FUNCTION_BLOCK EQUIP_TRIManager (* Composite Function Block Type *)
  (* Standard: 61499-2 *)
  (* Version 0.0, 08/01/2026, Schneider Electric, template *)
  PACKAGE Main;
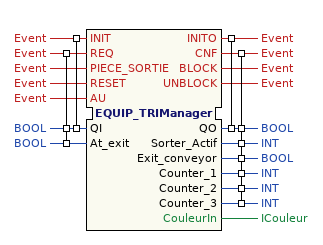
  EVENT_INPUT
    INIT WITH QI; (* Initialization Request *)
    REQ WITH QI, At_exit; (* Normal Execution Request *)
    PIECE_SORTIE;
    RESET; (* Reset compteurs et etapes *)
    AU; (* Arret urgence *)
  END_EVENT
  EVENT_OUTPUT
    INITO WITH QO; (* Initialization Confirm *)
    CNF WITH QO, Sorter_Actif, Exit_conveyor, Counter_1, Counter_2, Counter_3; (* Execution Confirmation *)
    BLOCK; (* Bloquer le convoyeur d'entrée *)
    UNBLOCK; (* Débloquer le convoyeur d'entrée *)
  END_EVENT
  VAR_INPUT
    QI : BOOL; (* Input event qualifier *)
    At_exit : BOOL; (* Capteur sortie - TRUE si piece presente *)
  END_VAR
  VAR_OUTPUT
    QO : BOOL; (* Output event qualifier *)
    Sorter_Actif : INT;
    Exit_conveyor : BOOL;
    Counter_1 : INT;
    Counter_2 : INT;
    Counter_3 : INT;
  END_VAR
  PLUGS
    CouleurIn : ICouleur; (* Entrée couleur *)
  END_PLUGS
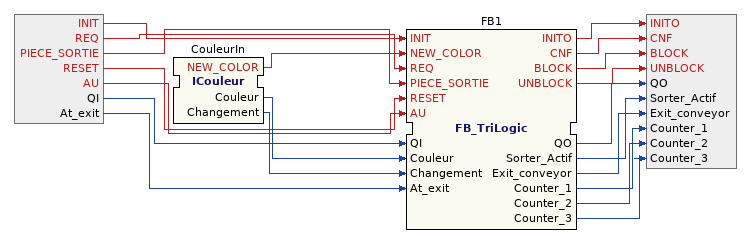
  FBS
    FB1 : FB_TriLogic;
  END_FBS
  EVENT_CONNECTIONS
    FB1.INITO TO INITO;
    FB1.CNF TO CNF;
    FB1.BLOCK TO BLOCK;
    FB1.UNBLOCK TO UNBLOCK;
    INIT TO FB1.INIT;
    REQ TO FB1.REQ;
    CouleurIn.NEW_COLOR TO FB1.NEW_COLOR;
    PIECE_SORTIE TO FB1.PIECE_SORTIE;
    RESET TO FB1.RESET;
    AU TO FB1.AU;
  END_CONNECTIONS
  DATA_CONNECTIONS
    FB1.QO TO QO;
    FB1.Exit_conveyor TO Exit_conveyor;
    FB1.Sorter_Actif TO Sorter_Actif;
    FB1.Counter_1 TO Counter_1;
    FB1.Counter_2 TO Counter_2;
    FB1.Counter_3 TO Counter_3;
    CouleurIn.Couleur TO FB1.Couleur;
    CouleurIn.Changement TO FB1.Changement;
    QI TO FB1.QI;
    At_exit TO FB1.At_exit;
  END_CONNECTIONS
END_FUNCTION_BLOCK
